(* PLC project Pump Control Example, CONTROLLINO GmbH CONTROLLINO MAXI Automation 0.1.0, author Firmware Team *)
(* stored: creationDateTime 2022-06-29T09:04:32, contentDescription Pump control example for CONTROLLINO MAXI Automation Outputs: DO0 -> %QX0.0 -> Process running/emergency indicator DO1 -> %QX0.1 -> Pump working indicator DO2 -> %QX0.2 -> High level indicator DO3 -> %QX0.3 -> Low level indicator R0 -> %QX1.0 -> Control pump contactor coil Inputs: AI2 -> %IX0.0 -> NO Pump contactor auxiliary contact AI3 -> %IX0.1 -> NO High level sensor contact AI4 -> %IX0.2 -> NO Low level sensor contact AI5 -> %IX0.3 -> NC Pump magnetothermic protection auxiliary contact AI6 -> %IX0.4 -> NO Start button AI7 -> %IX0.5 -> NC Stop button Behavior: The start button starts the process, the pump will try to maintain the level between the low and high levels. The stop button stops the process. The pump turns on when the level is lower than the low level sensor and stops when it reaches the high level. The low level indicator will blink with a period of N milliseconds in case of critical level, meaning that the level is bellow low level sensor. The emergency condition stops the process and occurs when the magnetothermic pump protection activates its auxiliary contact, or the pump feedback from pump contactor auxiliary contact is not recieved after N seconds, or also when the pump does not reach the desired level after N seconds. In an emergency condition, the emergency indicator blink with a period of N milliseconds. After the emergency condition, the start button must be pressed to reset the emergency condition and try to restart the process, also the stop button resets the emergency condition. MIT License Copyright (c) 2016-2022 CONTROLLINO GmbH Permission is hereby granted, free of charge, to any person obtaining a copy of this software and associated documentation files (the "Software"), to deal in the Software without restriction, including without limitation the rights to use, copy, modify, merge, publish, distribute, sublicense, and/or sell copies of the Software, and to permit persons to whom the Software is furnished to do so, subject to the following conditions: The above copyright notice and this permission notice shall be included in all copies or substantial portions of the Software. THE SOFTWARE IS PROVIDED "AS IS", WITHOUT WARRANTY OF ANY KIND, EXPRESS OR IMPLIED, INCLUDING BUT NOT LIMITED TO THE WARRANTIES OF MERCHANTABILITY, FITNESS FOR A PARTICULAR PURPOSE AND NONINFRINGEMENT. IN NO EVENT SHALL THE AUTHORS OR COPYRIGHT HOLDERS BE LIABLE FOR ANY CLAIM, DAMAGES OR OTHER LIABILITY, WHETHER IN AN ACTION OF CONTRACT, TORT OR OTHERWISE, ARISING FROM, OUT OF OR IN CONNECTION WITH THE SOFTWARE OR THE USE OR OTHER DEALINGS IN THE SOFTWARE. CONTROLLINO - First software open-source PLC (ARDUINO compatible) https://controllino.com/ https://github.com/CONTROLLINO-PLC/OpenPLC_examples https://www.arduino.cc/ author: CONTROLLINO firmware team version: 0.1.0, modificationDateTime 2022-07-14T12:27:13, version 0.1.0 *)

PROGRAM inputs
  VAR
    AI2 AT %IX0.0 : BOOL;
    AI3 AT %IX0.1 : BOOL;
    AI4 AT %IX0.2 : BOOL;
    AI5 AT %IX0.3 : BOOL;
    AI6 AT %IX0.4 : BOOL;
    AI7 AT %IX0.5 : BOOL;
  END_VAR
  VAR_EXTERNAL
    PUMP_ON : BOOL;
    HIGH_LEVEL : BOOL;
    LOW_LEVEL : BOOL;
    PUMP_PROTECTION_NC : BOOL;
    START : BOOL;
    STOP_NC : BOOL;
  END_VAR

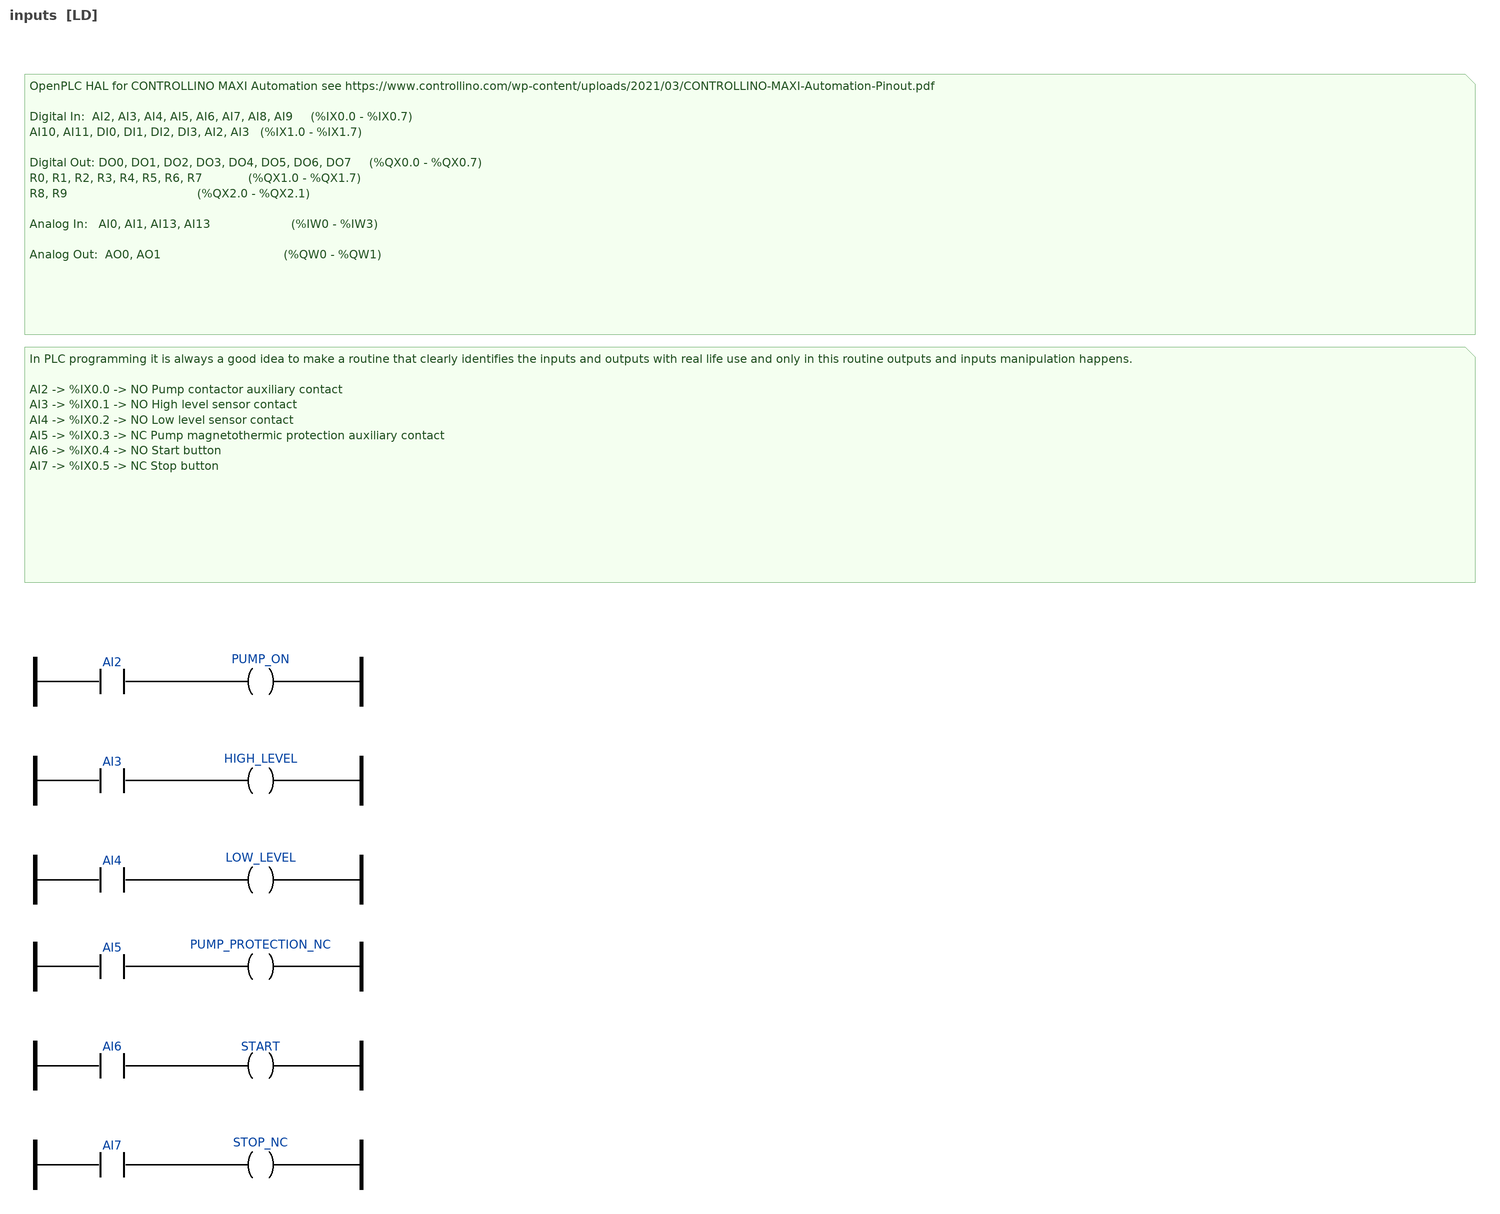
(* LD diagram, written out as Structured Text *)
(* OpenPLC HAL for CONTROLLINO MAXI Automation see https://www.controllino.com/wp-content/uploads/2021/03/CONTROLLINO-MAXI-Automation-Pinout.pdf

Digital In:  AI2, AI3, AI4, AI5, AI6, AI7, AI8, AI9     (%IX0.0 - %IX0.7)
             AI10, AI11, DI0, DI1, DI2, DI3, AI2, AI3   (%IX1.0 - %IX1.7)

Digital Out: DO0, DO1, DO2, DO3, DO4, DO5, DO6, DO7     (%QX0.0 - %QX0.7)
             R0, R1, R2, R3, R4, R5, R6, R7             (%QX1.0 - %QX1.7)
             R8, R9                                     (%QX2.0 - %QX2.1)

Analog In:   AI0, AI1, AI13, AI13                       (%IW0 - %IW3)

Analog Out:  AO0, AO1                                   (%QW0 - %QW1) *)
(* In PLC programming it is always a good idea to make a routine that clearly identifies the inputs and outputs with real life use and only in this routine outputs and inputs manipulation happens.

AI2 -> %IX0.0 -> NO Pump contactor auxiliary contact
AI3 -> %IX0.1 -> NO High level sensor contact
AI4 -> %IX0.2 -> NO Low level sensor contact
AI5 -> %IX0.3 -> NC Pump magnetothermic protection auxiliary contact
AI6 -> %IX0.4 -> NO Start button
AI7 -> %IX0.5 -> NC Stop button *)
PUMP_ON := AI2;
HIGH_LEVEL := AI3;
LOW_LEVEL := AI4;
PUMP_PROTECTION_NC := AI5;
START := AI6;
STOP_NC := AI7;
END_PROGRAM

PROGRAM control
  VAR_EXTERNAL
    START : BOOL;
    STOP_NC : BOOL;
    EMERGENCY : BOOL;
    HIGH_LEVEL : BOOL;
    LOW_LEVEL : BOOL;
    PUMP_CONTROL : BOOL;
    RUN : BOOL;
  END_VAR

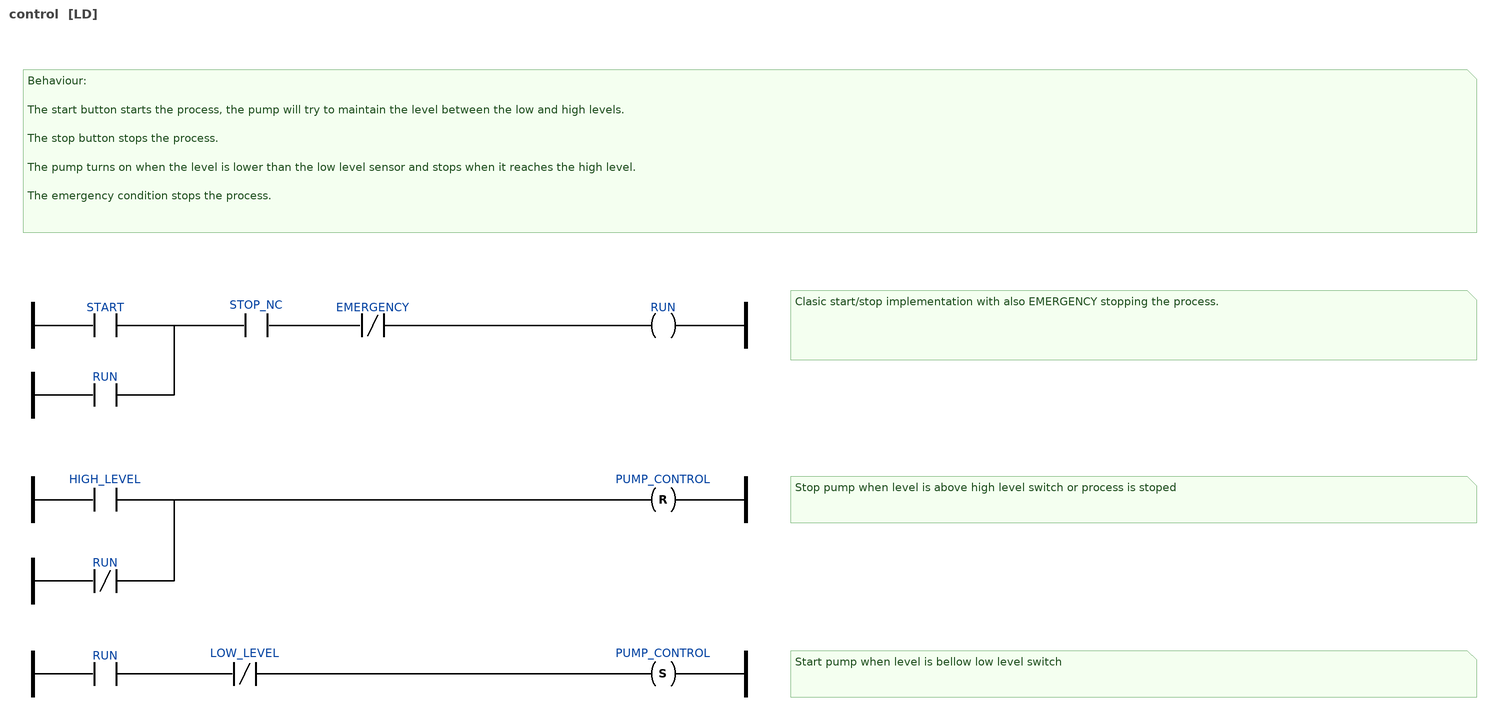
(* LD diagram, written out as Structured Text *)
(* Behaviour:

The start button starts the process, the pump will try to maintain the level between the low and high levels.

The stop button stops the process.

The pump turns on when the level is lower than the low level sensor and stops when it reaches the high level.

The emergency condition stops the process. *)
(* Clasic start/stop implementation with also EMERGENCY stopping the process. *)
RUN := (START OR RUN) AND STOP_NC AND NOT EMERGENCY;
(* Stop pump when level is above high level switch or process is stoped *)
IF HIGH_LEVEL OR NOT RUN THEN PUMP_CONTROL := FALSE; END_IF;
(* Start pump when level is bellow low level switch *)
IF RUN AND NOT LOW_LEVEL THEN PUMP_CONTROL := TRUE; END_IF;
END_PROGRAM

PROGRAM outputs
  VAR
    DO0 AT %QX0.0 : BOOL;
    DO1 AT %QX0.1 : BOOL;
    DO2 AT %QX0.2 : BOOL;
    DO3 AT %QX0.3 : BOOL;
    R0 AT %QX1.0 : BOOL;
  END_VAR
  VAR_EXTERNAL
    PUMP_ON : BOOL;
    HIGH_LEVEL : BOOL;
    LOW_LEVEL : BOOL;
    PUMP_CONTROL : BOOL;
    EMERGENCY : BOOL;
    RUN : BOOL;
  END_VAR
  VAR
    T_BLINK : TIME := T#500ms;
    EMERGENCY_INDICATOR : BOOL;
    CRITICAL_LEVEL_INDICATOR : BOOL;
    TON0 : TON;
    TON1 : TON;
    TON2 : TON;
    TON3 : TON;
  END_VAR

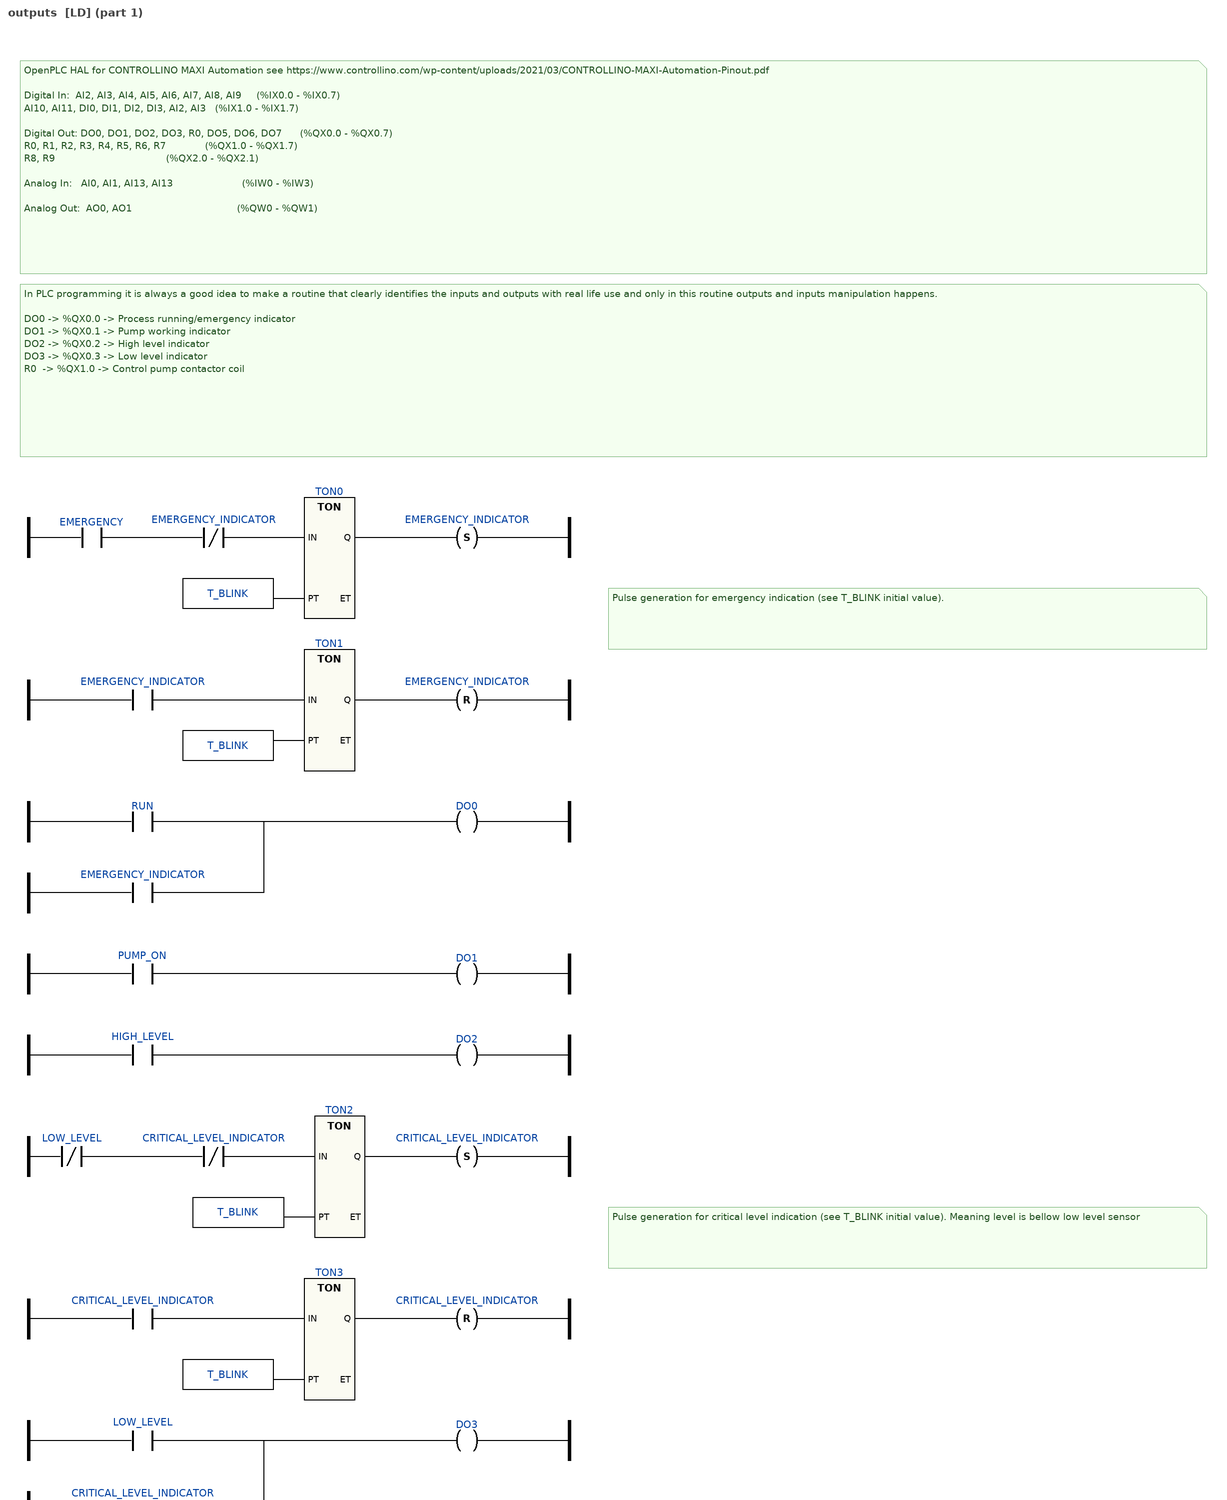
(* LD diagram, written out as Structured Text *)
(* OpenPLC HAL for CONTROLLINO MAXI Automation see https://www.controllino.com/wp-content/uploads/2021/03/CONTROLLINO-MAXI-Automation-Pinout.pdf

Digital In:  AI2, AI3, AI4, AI5, AI6, AI7, AI8, AI9     (%IX0.0 - %IX0.7)
             AI10, AI11, DI0, DI1, DI2, DI3, AI2, AI3   (%IX1.0 - %IX1.7)

Digital Out: DO0, DO1, DO2, DO3, R0, DO5, DO6, DO7      (%QX0.0 - %QX0.7)
             R0, R1, R2, R3, R4, R5, R6, R7             (%QX1.0 - %QX1.7)
             R8, R9                                     (%QX2.0 - %QX2.1)

Analog In:   AI0, AI1, AI13, AI13                       (%IW0 - %IW3)

Analog Out:  AO0, AO1                                   (%QW0 - %QW1) *)
(* In PLC programming it is always a good idea to make a routine that clearly identifies the inputs and outputs with real life use and only in this routine outputs and inputs manipulation happens.

DO0 -> %QX0.0 -> Process running/emergency indicator
DO1 -> %QX0.1 -> Pump working indicator
DO2 -> %QX0.2 -> High level indicator
DO3 -> %QX0.3 -> Low level indicator
R0  -> %QX1.0 -> Control pump contactor coil *)
TON0(IN := EMERGENCY AND NOT EMERGENCY_INDICATOR, PT := T_BLINK);
IF TON0.Q THEN EMERGENCY_INDICATOR := TRUE; END_IF;
(* Pulse generation for emergency indication (see T_BLINK initial value). *)
TON1(IN := EMERGENCY_INDICATOR, PT := T_BLINK);
IF TON1.Q THEN EMERGENCY_INDICATOR := FALSE; END_IF;
DO0 := RUN OR EMERGENCY_INDICATOR;
DO1 := PUMP_ON;
DO2 := HIGH_LEVEL;
TON2(IN := NOT LOW_LEVEL AND NOT CRITICAL_LEVEL_INDICATOR, PT := T_BLINK);
IF TON2.Q THEN CRITICAL_LEVEL_INDICATOR := TRUE; END_IF;
(* Pulse generation for critical level indication (see T_BLINK initial value). Meaning level is bellow low level sensor *)
TON3(IN := CRITICAL_LEVEL_INDICATOR, PT := T_BLINK);
IF TON3.Q THEN CRITICAL_LEVEL_INDICATOR := FALSE; END_IF;
DO3 := LOW_LEVEL OR CRITICAL_LEVEL_INDICATOR;
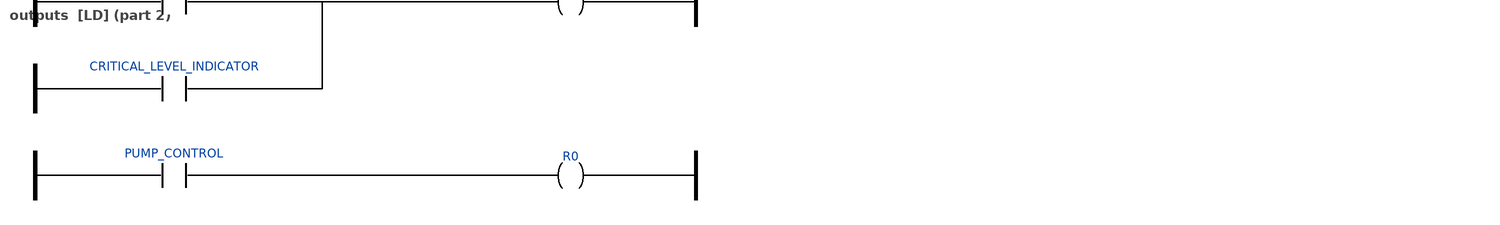
R0 := PUMP_CONTROL;
END_PROGRAM

PROGRAM emergency_check
  VAR_EXTERNAL
    PUMP_PROTECTION_NC : BOOL;
    PUMP_ON : BOOL;
    PUMP_CONTROL : BOOL;
    HIGH_LEVEL : BOOL;
    LOW_LEVEL : BOOL;
    EMERGENCY : BOOL;
    RUN : BOOL;
    STOP_NC : BOOL;
  END_VAR
  VAR
    T_ERROR_PUMP_ON : TIME := T#5s;
    T_ERROR_LEVEL : TIME := T#10s;
    ERROR_PUMP_PROTECTION : BOOL;
    ERROR_PUMP_ON : BOOL;
    ERROR_LEVEL_LOW : BOOL;
    ERROR_LEVEL_HIGH : BOOL;
    TON0 : TON;
    TON1 : TON;
    TON2 : TON;
  END_VAR
  VAR  (* added by the conversion: wires and edge detectors of the diagram *)
    R_TRIG1 : R_TRIG;
    R_TRIG2 : R_TRIG;
    R_TRIG3 : R_TRIG;
    R_TRIG4 : R_TRIG;
    R_TRIG5 : R_TRIG;
    F_TRIG6 : F_TRIG;
  END_VAR

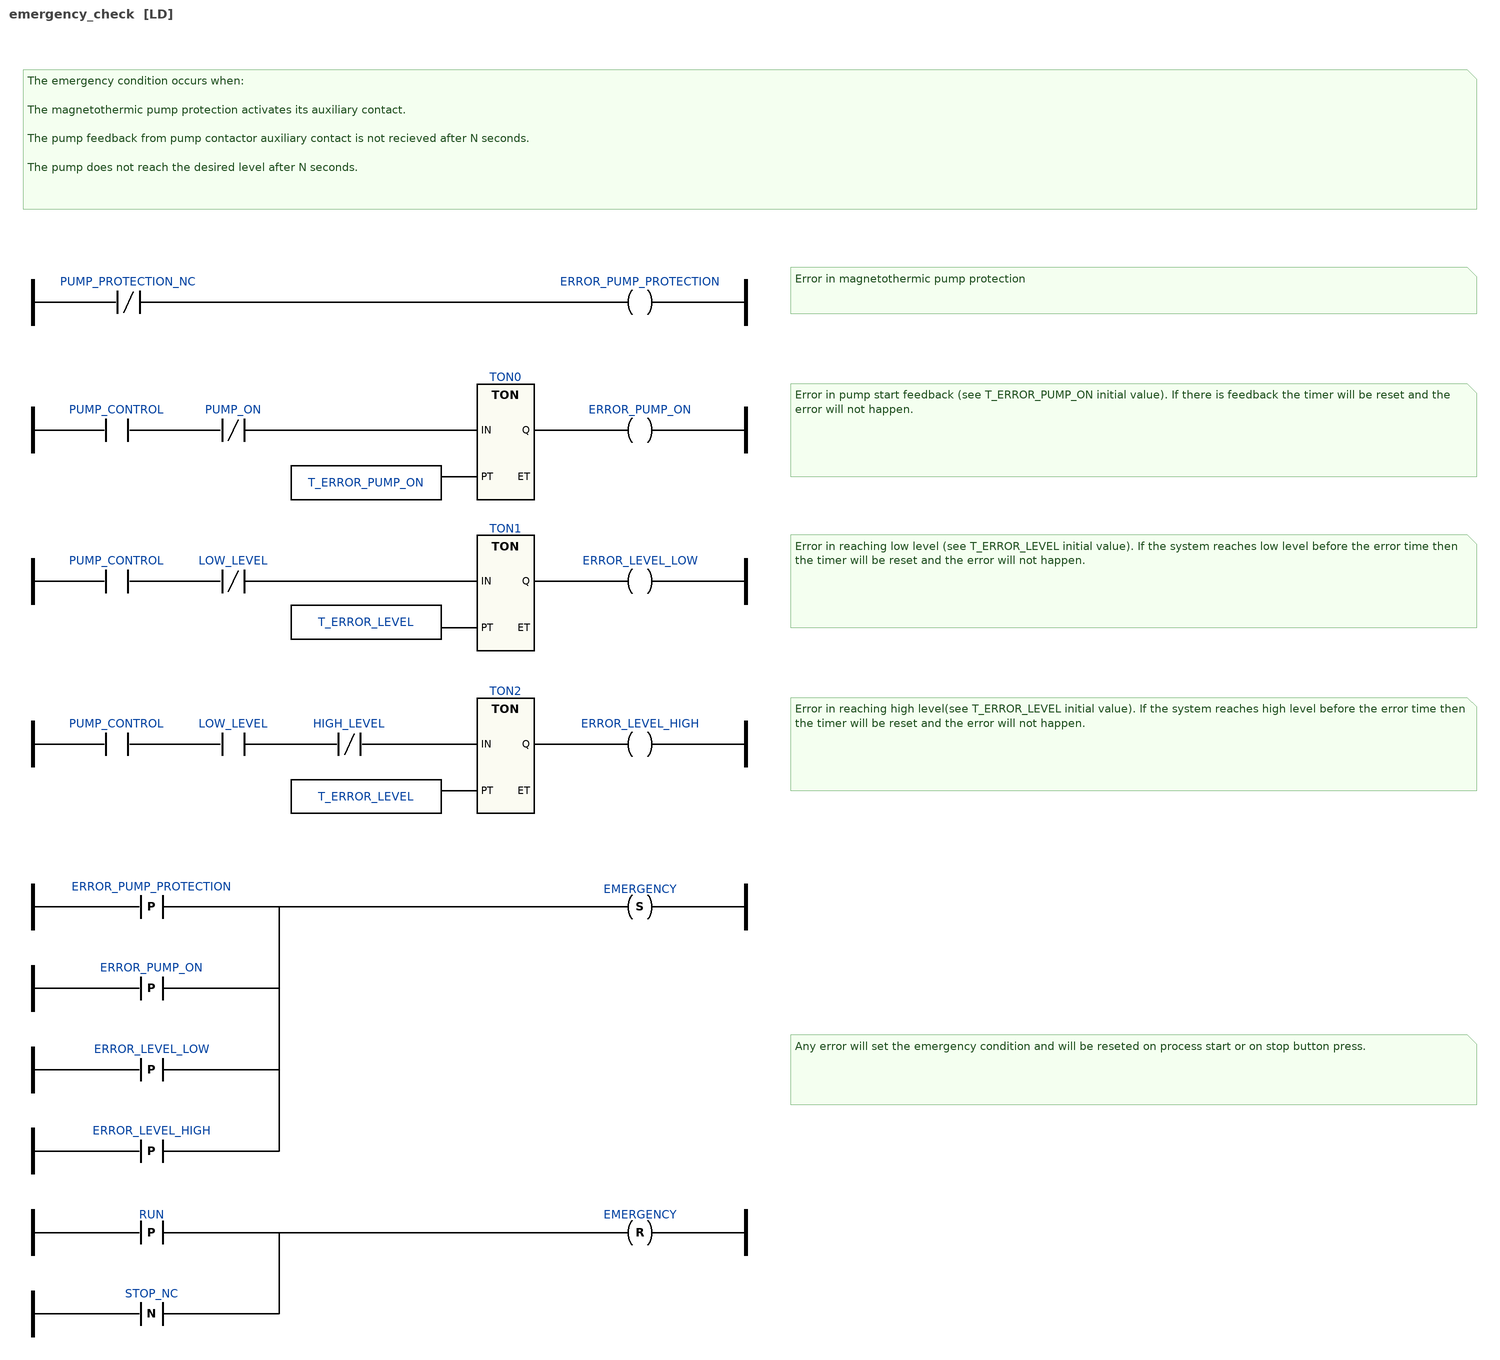
(* LD diagram, written out as Structured Text *)
(* The emergency condition occurs when:

    The magnetothermic pump protection activates its auxiliary contact.

    The pump feedback from pump contactor auxiliary contact is not recieved after N seconds.

    The pump does not reach the desired level after N seconds. *)
(* Error in magnetothermic pump protection *)
ERROR_PUMP_PROTECTION := NOT PUMP_PROTECTION_NC;
(* Error in pump start feedback (see T_ERROR_PUMP_ON initial value). If there is feedback the timer will be reset and the error will not happen. *)
TON0(IN := PUMP_CONTROL AND NOT PUMP_ON, PT := T_ERROR_PUMP_ON);
ERROR_PUMP_ON := TON0.Q;
(* Error in reaching low level (see T_ERROR_LEVEL initial value). If the system reaches low level before the error time then the timer will be reset and the error will not happen. *)
TON1(IN := PUMP_CONTROL AND NOT LOW_LEVEL, PT := T_ERROR_LEVEL);
ERROR_LEVEL_LOW := TON1.Q;
(* Error in reaching high level(see T_ERROR_LEVEL initial value). If the system reaches high level before the error time then the timer will be reset and the error will not happen. *)
TON2(IN := PUMP_CONTROL AND LOW_LEVEL AND NOT HIGH_LEVEL, PT := T_ERROR_LEVEL);
ERROR_LEVEL_HIGH := TON2.Q;
R_TRIG1(CLK := ERROR_PUMP_PROTECTION);
R_TRIG2(CLK := ERROR_PUMP_ON);
R_TRIG3(CLK := ERROR_LEVEL_LOW);
R_TRIG4(CLK := ERROR_LEVEL_HIGH);
IF R_TRIG1.Q OR R_TRIG2.Q OR R_TRIG3.Q OR R_TRIG4.Q THEN EMERGENCY := TRUE; END_IF;
(* Any error will set the emergency condition and will be reseted on process start or on stop button press. *)
R_TRIG5(CLK := RUN);
F_TRIG6(CLK := STOP_NC);
IF R_TRIG5.Q OR F_TRIG6.Q THEN EMERGENCY := FALSE; END_IF;
END_PROGRAM

CONFIGURATION Config0
  RESOURCE Res0 ON PLC
    VAR_GLOBAL
      PUMP_ON : BOOL;
      HIGH_LEVEL : BOOL;
      LOW_LEVEL : BOOL;
      PUMP_PROTECTION_NC : BOOL;
      START : BOOL;
      STOP_NC : BOOL;
      PUMP_CONTROL : BOOL;
      EMERGENCY : BOOL;
      RUN : BOOL;
    END_VAR
    TASK task0(INTERVAL := T#20ms, PRIORITY := 0);
    PROGRAM instance0 WITH task0 : inputs;
    PROGRAM instance1 WITH task0 : control;
    PROGRAM instance2 WITH task0 : outputs;
    PROGRAM instance3 WITH task0 : emergency_check;
  END_RESOURCE
END_CONFIGURATION
